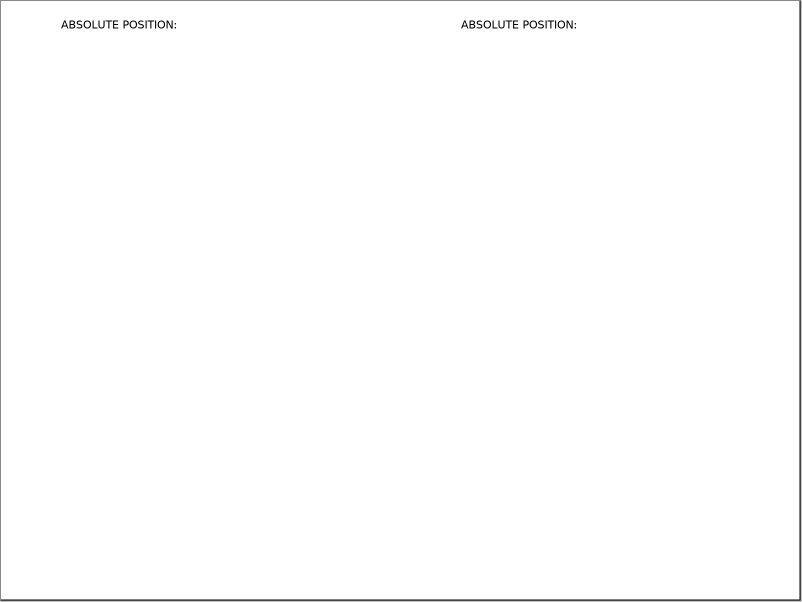
VISUALIZATION F03_Read_Status  // 802x602
    Rectangle (0,0 800x600)
    Label (10,10 170x30), "ABSOLUTE POSITION:"
    Label (410,10 170x30), "ABSOLUTE POSITION:"
END_VISUALIZATION

(* stored: Version 1.1.0.1, ProductVersion 3.1.4022.7
   Visu F03_Read_Status: Id {2313532c-5e9e-479a-81cc-67ae24a61e1a} *)
